FUNCTION_BLOCK AI_INT_TO_I (* Composite FB for convert INT to AI *)
  (* Standard: 61499-2; Description: Copyright (c) 2026 HR Agrartechnik GmbH This program and the accompanying materials are made available under the terms of the Eclipse Public License 2.0 which is available at https://www.eclipse.org/legal/epl-2.0/ SPDX-License-Identifier: EPL-2.0 *)
  (* Version 1.0, 2026-01-17, Franz Hoepfinger, HR Agrartechnik GmbH *)
  PACKAGE adapter::conversion::unidirectional;
  IMPORT eclipse4diac::core::TypeHash;
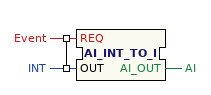
  EVENT_INPUT
    REQ WITH OUT; (* Request to Adapter *)
  END_EVENT
  VAR_INPUT
    OUT : INT;
  END_VAR
  PLUGS
    AI_OUT : adapter::types::unidirectional::AI; (* Adapter Output *)
  END_PLUGS
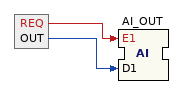
  EVENT_CONNECTIONS
    REQ TO AI_OUT.E1;
  END_CONNECTIONS
  DATA_CONNECTIONS
    OUT TO AI_OUT.D1;
  END_CONNECTIONS
END_FUNCTION_BLOCK
